INTERFACE I_AsyncResponseManager

METHOD TryConvertResponseToAsyncResponseSessionData : BOOL
VAR_INPUT
	Response : I_ServerResponse;
	RetryDelayInMs : UDINT;
	Destination : REFERENCE TO I_AsyncResponseSessionData;
END_VAR
END_METHOD

METHOD PUBLIC TryHandleIncomingRequest : BOOL
VAR_INPUT
	Request : I_Request;
	Response : I_ServerResponse;
END_VAR
END_METHOD

END_INTERFACE

(* stored: Version 1.1.0.1, ProductVersion 3.1.4026.13
   Itf I_AsyncResponseManager: Id {e66426b4-8976-41c4-8618-3a237a7a5dc6}
   Method TryConvertResponseToAsyncResponseSessionData: Id {1c256675-c6f3-4a69-abe1-023a0168c972}
   Method TryHandleIncomingRequest: Id {0f01b17a-9511-4c12-b684-a1173a95c487} *)
